// TIA Portal V18 export
FUNCTION_BLOCK "wwwMain"   // FB9, FBD
{ S7_Optimized_Access := 'TRUE' }
VERSION : 0.1
// stored: AutoNumber true, IsIECCheckEnabled false, IsRetainMemResEnabled false, MemoryReserve 100, SetENOAutomatically false, UDAEnableTagReadback false
   VAR_TEMP
      RET_VAL : Int;
      temp : Int;
   END_VAR
BEGIN

REGION Network 1: ActualValues -> Web data
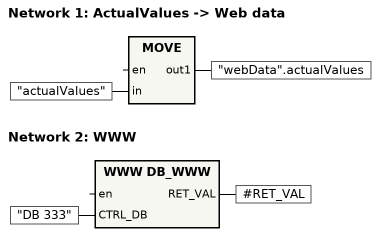
   "webData".actualValues := "actualValues";
END_REGION

REGION Network 2: WWW
   #RET_VAL := WWW(CTRL_DB := "DB 333");
END_REGION
END_FUNCTION_BLOCK
